(* Logix 5000 project; controller Turck_IOLink_All_Full_AOIs_V0_1 vendor 1 type 14 code 176 rev 32.11; software revision 32.00 *)

TASK MainTask (continuous, watchdog 500 ms) : MainProgram
TASK SafetyTask (periodic, rate 20 ms, priority 10, watchdog 20 ms, safety) : SafetyProgram

MODULES
   Local : vendor 1 type 14 code 176 (Compact 0, rev 32.11)
END_MODULES

TYPE Generic_16_Words :
STRUCT
   Data : INT[16];
END_STRUCT
END_TYPE

TYPE Turck_IOLink_Common_Data :
STRUCT
   Read : BOOL;   // For internal use to integrate IOLRead and IOWrite with IOLService
   Write : BOOL;   // For internal use to integrate IOLRead and IOWrite with IOLService
   Reset : BOOL;   // For internal use to integrate IOLRead and IOWrite with IOLService
   Done : BOOL;   // For internal use to integrate IOLRead and IOWrite with IOLService
   Error : BOOL;   // For internal use to integrate IOLRead and IOWrite with IOLService
   Port_in_Use : SINT;   // Each bit is set to show that a port is in use. If it's not in use the port diagnostics will be disabled so IO-Link can still be used but won't throw a red light if no device plugged
   Port : INT;   // For internal use to integrate IOLRead and IOWrite with IOLService
   Index : INT;   // For internal use to integrate IOLRead and IOWrite with IOLService
   SubIndex : INT;   // For internal use to integrate IOLRead and IOWrite with IOLService
   Length : INT;   // For internal use to integrate IOLRead and IOWrite with IOLService
   TicketNum : INT;   // For internal use to integrate IOLRead and IOWrite with IOLService
   Status : INT;   // For internal use to integrate IOLRead and IOWrite with IOLService
   NextTicketNum : INT;   // For internal use to integrate IOLRead and IOWrite with IOLService
   ReceiveData : SINT[255];   // For internal use to integrate IOLRead and IOWrite with IOLService
   SendData : SINT[145];   // For internal use to integrate IOLRead and IOWrite with IOLService
   Vendor_IDs : INT[8];
   Device_IDs : DINT[8];
   WriteData : DINT;
   Process_Input_Data : Generic_16_Words[8];
   Process_Output_Data : Generic_16_Words[8];
END_STRUCT
END_TYPE

TYPE Universal_IOLink_Info :
STRUCT
   Vendor_Name : STRING;   // Index 16
   Vendor_Text : STRING;   // Index 17
   Product_Name : STRING;   // Index 18
   Product_ID : STRING;   // Index 19
   Product_Text : STRING;   // Index 20
   Serial_Number : STRING;   // Index 21
   Hardware_Revision : STRING;   // Index 22
   Firmware_Revision : STRING;   // Index 23
   Application_Specific_Tag : STRING;   // Index 24
   Function_Tag : STRING;   // Index 25
   Location_Tag : STRING;   // Index 26
   Application_Specific_Tag_Requested : STRING;
END_STRUCT
END_TYPE

ADD_ON_INSTRUCTION Banner_K50_Pro_Advanced_Mode_Full   (* revision 1.0 *)
VAR_INPUT
   Touch_Sensitivity : SINT := 1; {access None}   // Index 82 - Subindex 1 - 0 = Low, 1 = Standard, 2 = High (Default = 1)
   Touch_Function : BOOL;   // Index 82 - Subindex 2 - 0 = Momentary, 1 = Latched
   Touch_Mute_Enable : BOOL;   // Index 82 - Subindex 3 - 0 = Off, 1 = On
   Touch_On_Delay : SINT;   // Index 82 - Subindex 4 - 0-65535 ms
   Custom_Color_1_Red : INT;   // Index 88 - Subindex 1 - 0-255 Amount of Red
   Custom_Color_1_Green : INT;   // Index 88 - Subindex 2 - 0-255 Amount of Green
   Custom_Color_1_Blue : INT;   // Index 88 - Subindex 3 - 0-255 Amount of Blue
   Custom_Color_2_Red : INT;   // Index 89 - Subindex 1 - 0-255 Amount of Red
   Custom_Color_2_Green : INT;   // Index 89 - Subindex 2 - 0-255 - Amount of Green
   Custom_Color_2_Blue : INT;   // Index 89 - Subindex 3 - 0-255 - Amount of Blue
   Port : INT; {required}
END_VAR
VAR_IN_OUT
   Common_Data : Turck_IOLink_Common_Data; {required}
END_VAR
VAR_INPUT
   Animation_Type : SINT; {visible}   // 0 = Off 1 = Steady 2 = Flash 3 = Two Color Flash 4 = 50/50 5 = 50/50 Rotate 6 = Chase 7 = Intensity Sweep 8 = Color Sweep 9 = Sequence
   Animation_Direction : BOOL; {visible}   // 0 = CCW, 1 = CW
   Animation_Pattern : SINT; {visible}   // 0 = Flash, 1 = Strobe, 2 = Three Pulse, 3 = SOS, 4 = Random
   Animation_Speed : SINT; {visible}   // 0 = Slow, 1 = Medium, 2 = Fast, 3 = Custom
   Vibration_Feedback : SINT; {visible}   // 0 = Off, 1 = On, 2 = Animation Pattern
   Dynamic_Sequence : INT; {visible}   // 0-255
   Sequence_Start_Location : SINT; {visible}   // 0 = LED1 1 = LED2 2 = LED3 3 = LED4 4 = LED5 5 = LED6 6 = LED7 7 = LED8
   Color_1 : SINT; {visible}   // 0 = Green 1 = Red 2 = Orange 3 = Amber 4 = Yellow 5 = Lime Green 6 = Spring Green 7 = Cyan 8 = Sky Blue 9 = Blue 10 = Violet 11 = Magenta 12 = Rose 13 = White 14 = Custom1 15 = Custom2
   Color_1_Intensity : SINT; {visible}   // 0 = High, 1 = Medium, 2 = Low, 3 = Off, 4 = Custom
   Color_2 : SINT; {visible}   // 0 = Green 1 = Red 2 = Orange 3 = Amber 4 = Yellow 5 = Lime Green 6 = Spring Green 7 = Cyan 8 = Sky Blue 9 = Blue 10 = Violet 11 = Magenta 12 = Rose 13 = White 14 = Custom1 15 = Custom2
   Color_2_Intensity : SINT; {visible}   // 0 = High, 1 = Medium, 2 = Low, 3 = Off, 4 = Custom
END_VAR
VAR_OUTPUT
   Output_State : BOOL; {access Read Only, visible}   // 0 = Inactive, 1 = Active
   Wrong_or_Missing_Device : BOOL; {access Read Only, visible}
END_VAR
VAR
   Port_Less_One : INT; {access None}
   Port_Bit : SINT; {access None}
   Output_Mode : SINT; {access None}
   Done : DINT; {access None}
   Error : DINT; {access None}
   Active : DINT; {access None}
   Pending : DINT; {access None}
   Pending_or_Active : DINT; {access None}
   Write : DINT; {access None}
   WriteRequest : DINT; {access None}
   Custom_Color_1_Red_Prev : SINT; {access None}
   Custom_Color_1_Green_Prev : SINT; {access None}
   Custom_Color_1_Blue_Prev : SINT; {access None}
   Custom_Color_2_Green_Prev : SINT; {access None}
   StartupDone : BOOL; {access None}
   Read_ONS : DINT; {access None}
   Error_DINT : DINT; {access None}
   StartupCount : DINT; {access None}
   MyTicketNum : DINT[32]; {access None}
   ReadRequest : DINT; {access None}
   DoneCount : DINT; {access None}
   Status : DINT; {access None}
   ErrorCount : DINT; {access None}
   Write_ONS : DINT; {access None}
   Custom_Color_2_Blue_Prev : SINT; {access None}
   Custom_Color_2_Red_Prev : SINT; {access None}
   Device_Connected_ONS : DINT; {access None}
END_VAR

ROUTINE Logic   (* ladder *)
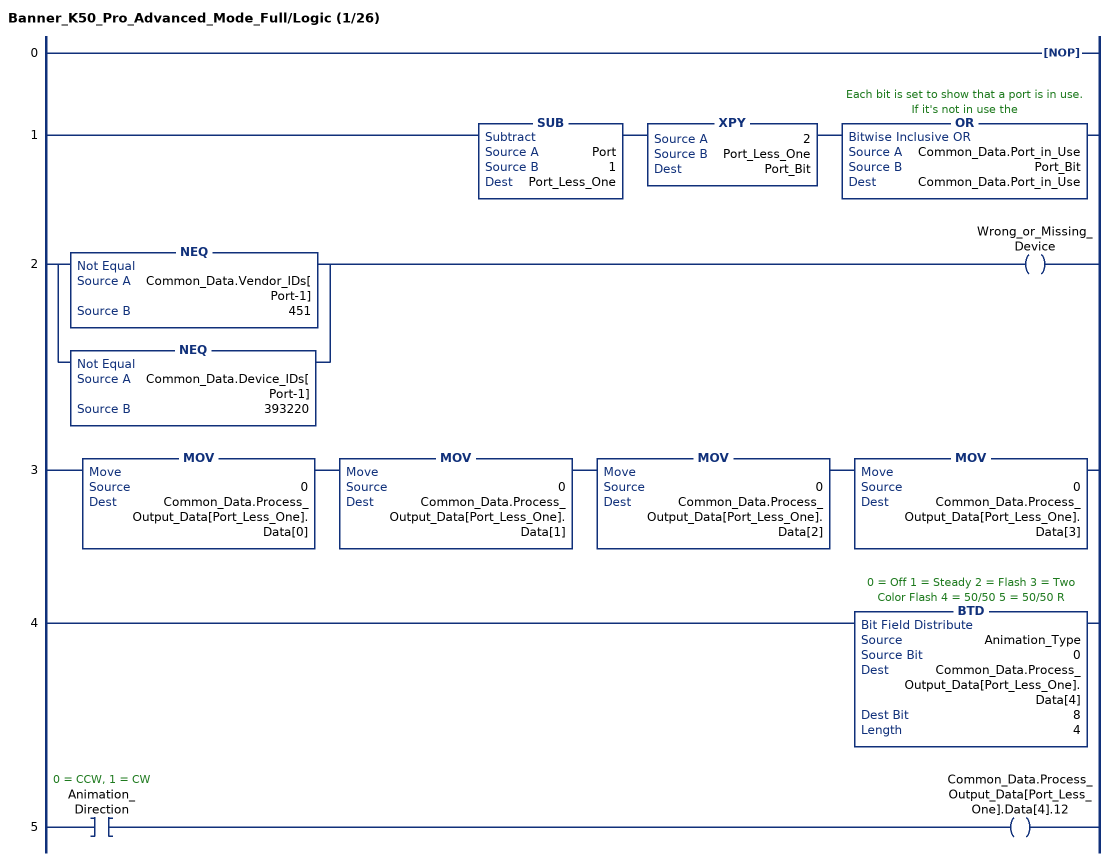
   0: NOP();
   1: SUB(Port,1,Port_Less_One)XPY(2,Port_Less_One,Port_Bit)OR(Common_Data.Port_in_Use,Port_Bit,Common_Data.Port_in_Use);
   2: [NEQ(Common_Data.Vendor_IDs[Port-1],451) ,NEQ(Common_Data.Device_IDs[Port-1],393220) ]OTE(Wrong_or_Missing_Device);
   3: MOV(0,Common_Data.Process_Output_Data[Port_Less_One].Data[0])MOV(0,Common_Data.Process_Output_Data[Port_Less_One].Data[1])MOV(0,Common_Data.Process_Output_Data[Port_Less_One].Data[2])MOV(0,Common_Data.Process_Output_Data[Port_Less_One].Data[3]);
   4: BTD(Animation_Type,0,Common_Data.Process_Output_Data[Port_Less_One].Data[4],8,4);
   5: XIC(Animation_Direction)OTE(Common_Data.Process_Output_Data[Port_Less_One].Data[4].12);
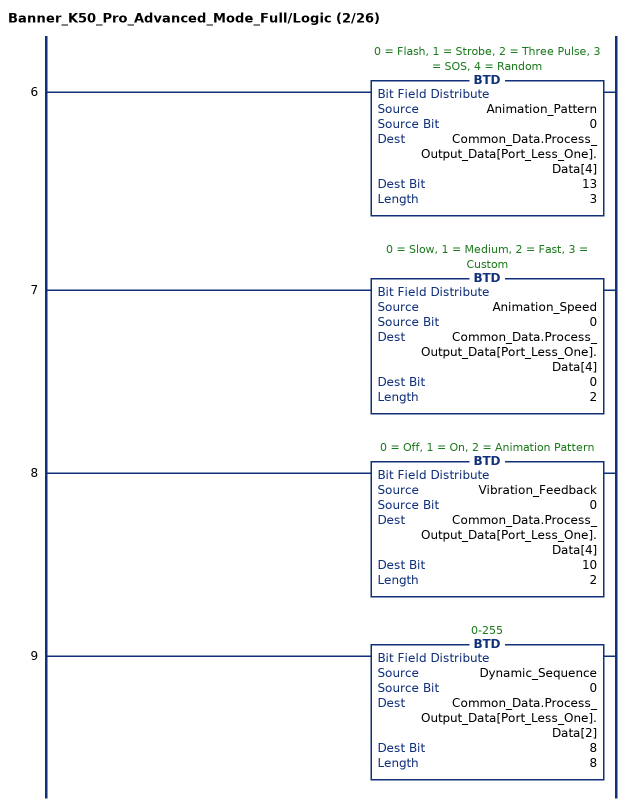
   6: BTD(Animation_Pattern,0,Common_Data.Process_Output_Data[Port_Less_One].Data[4],13,3);
   7: BTD(Animation_Speed,0,Common_Data.Process_Output_Data[Port_Less_One].Data[4],0,2);
   8: BTD(Vibration_Feedback,0,Common_Data.Process_Output_Data[Port_Less_One].Data[4],10,2);
   9: BTD(Dynamic_Sequence,0,Common_Data.Process_Output_Data[Port_Less_One].Data[2],8,8);
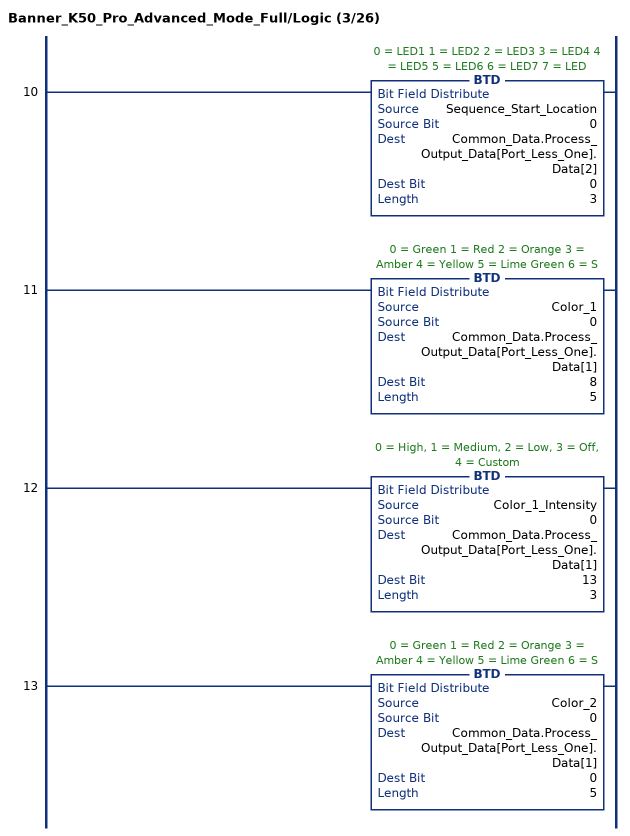
   10: BTD(Sequence_Start_Location,0,Common_Data.Process_Output_Data[Port_Less_One].Data[2],0,3);
   11: BTD(Color_1,0,Common_Data.Process_Output_Data[Port_Less_One].Data[1],8,5);
   12: BTD(Color_1_Intensity,0,Common_Data.Process_Output_Data[Port_Less_One].Data[1],13,3);
   13: BTD(Color_2,0,Common_Data.Process_Output_Data[Port_Less_One].Data[1],0,5);
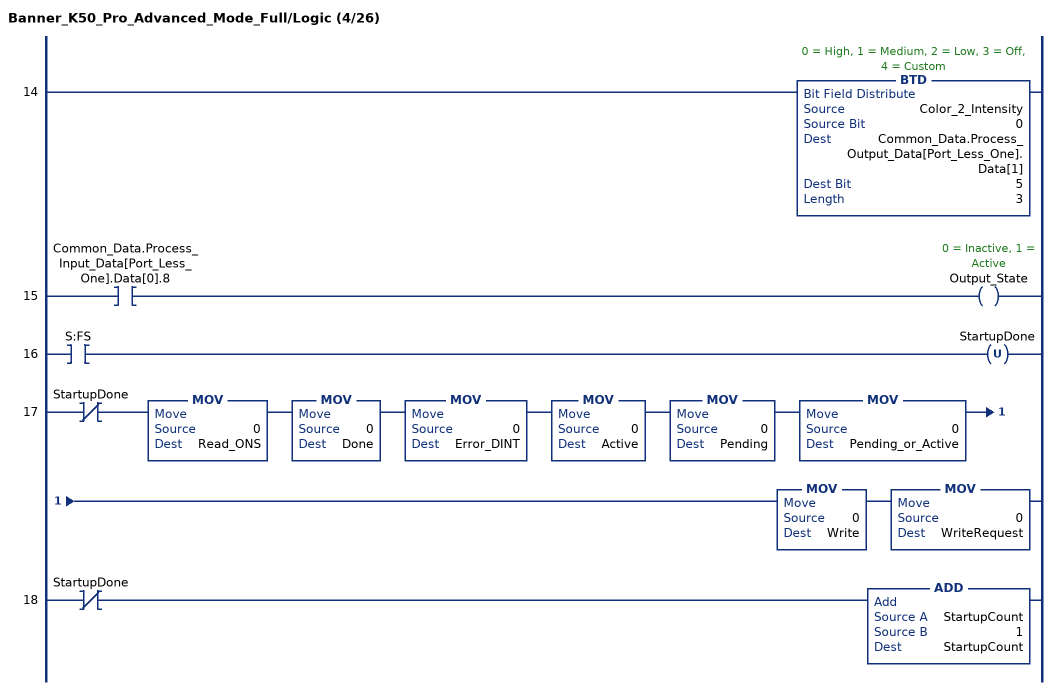
   14: BTD(Color_2_Intensity,0,Common_Data.Process_Output_Data[Port_Less_One].Data[1],5,3);
   15: XIC(Common_Data.Process_Input_Data[Port_Less_One].Data[0].8)OTE(Output_State);
   16: XIC(S:FS)OTU(StartupDone);
   17: XIO(StartupDone)MOV(0,Read_ONS)MOV(0,Done)MOV(0,Error_DINT)MOV(0,Active)MOV(0,Pending)MOV(0,Pending_or_Active)MOV(0,Write)MOV(0,WriteRequest);
   18: XIO(StartupDone)ADD(StartupCount,1,StartupCount);
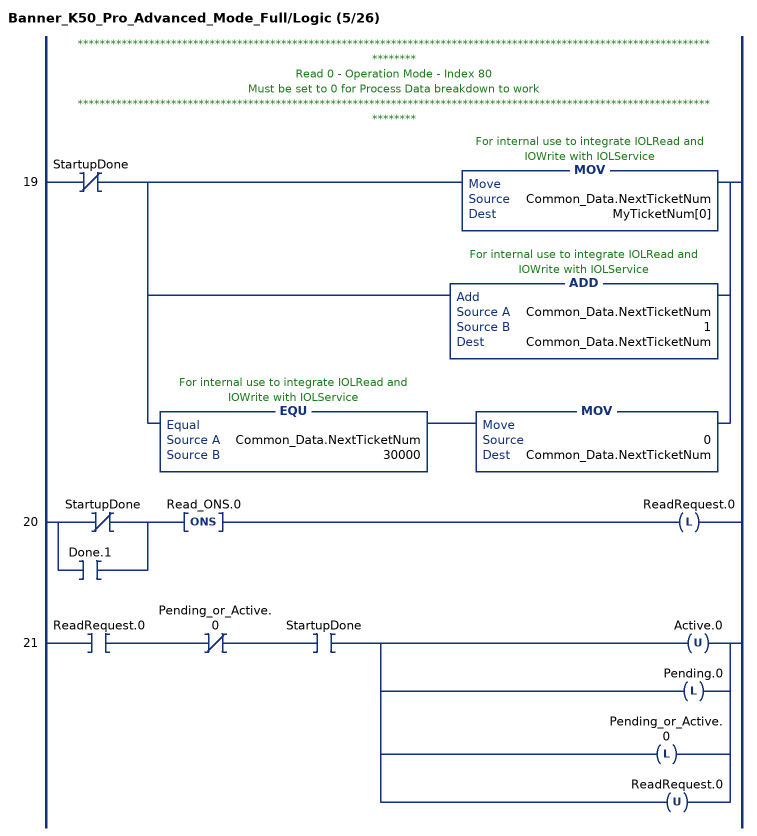
   // ***************************************************************************************************************************
   // Read 0 - Operation Mode - Index 80
   // Must be set to 0 for Process Data breakdown to work
   // ***************************************************************************************************************************
   19: XIO(StartupDone)[MOV(Common_Data.NextTicketNum,MyTicketNum[0]) ,ADD(Common_Data.NextTicketNum,1,Common_Data.NextTicketNum) ,EQU(Common_Data.NextTicketNum,30000) MOV(0,Common_Data.NextTicketNum) ];
   20: [XIO(StartupDone) ,XIC(Done.1) ]ONS(Read_ONS.0)OTL(ReadRequest.0);
   21: XIC(ReadRequest.0)XIO(Pending_or_Active.0)XIC(StartupDone)[OTU(Active.0) ,OTL(Pending.0) ,OTL(Pending_or_Active.0) ,OTU(ReadRequest.0) ];
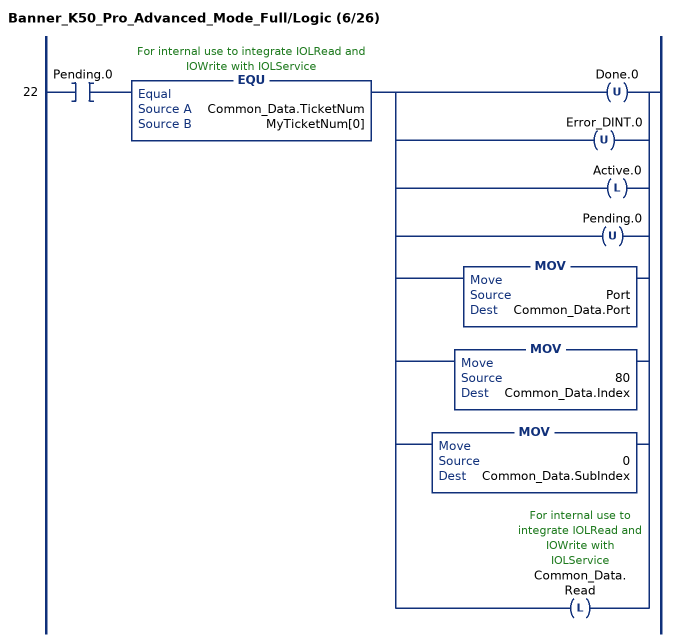
   22: XIC(Pending.0)EQU(Common_Data.TicketNum,MyTicketNum[0])[OTU(Done.0) ,OTU(Error_DINT.0) ,OTL(Active.0) ,OTU(Pending.0) ,MOV(Port,Common_Data.Port) ,MOV(80,Common_Data.Index) ,MOV(0,Common_Data.SubIndex) ,OTL(Common_Data.Read) ];
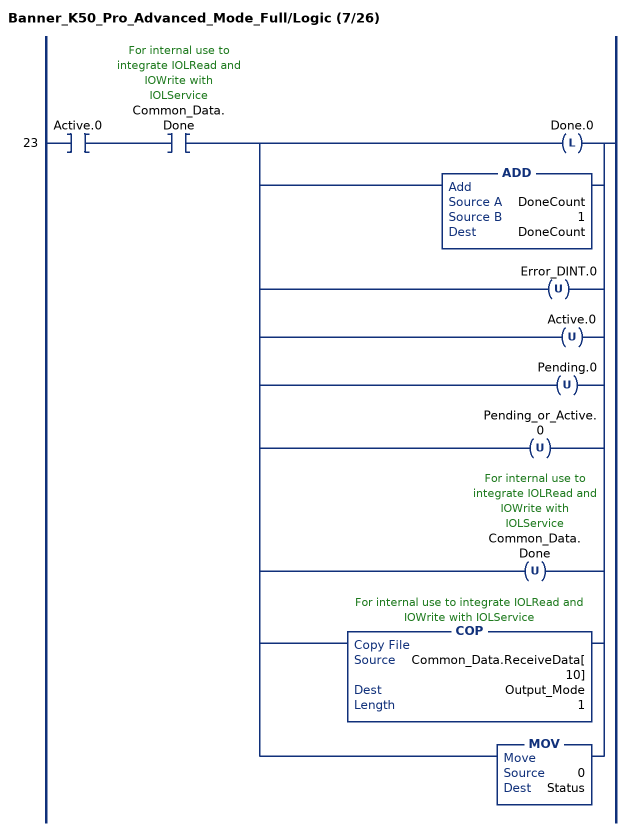
   23: XIC(Active.0)XIC(Common_Data.Done)[OTL(Done.0) ,ADD(DoneCount,1,DoneCount) ,OTU(Error_DINT.0) ,OTU(Active.0) ,OTU(Pending.0) ,OTU(Pending_or_Active.0) ,OTU(Common_Data.Done) ,COP(Common_Data.ReceiveData[10],Output_Mode,1) ,MOV(0,Status) ];
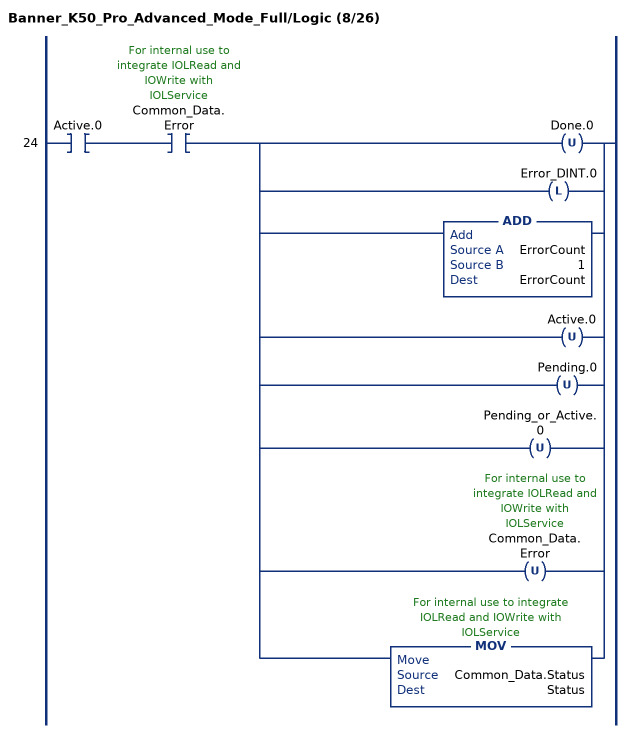
   24: XIC(Active.0)XIC(Common_Data.Error)[OTU(Done.0) ,OTL(Error_DINT.0) ,ADD(ErrorCount,1,ErrorCount) ,OTU(Active.0) ,OTU(Pending.0) ,OTU(Pending_or_Active.0) ,OTU(Common_Data.Error) ,MOV(Common_Data.Status,Status) ];
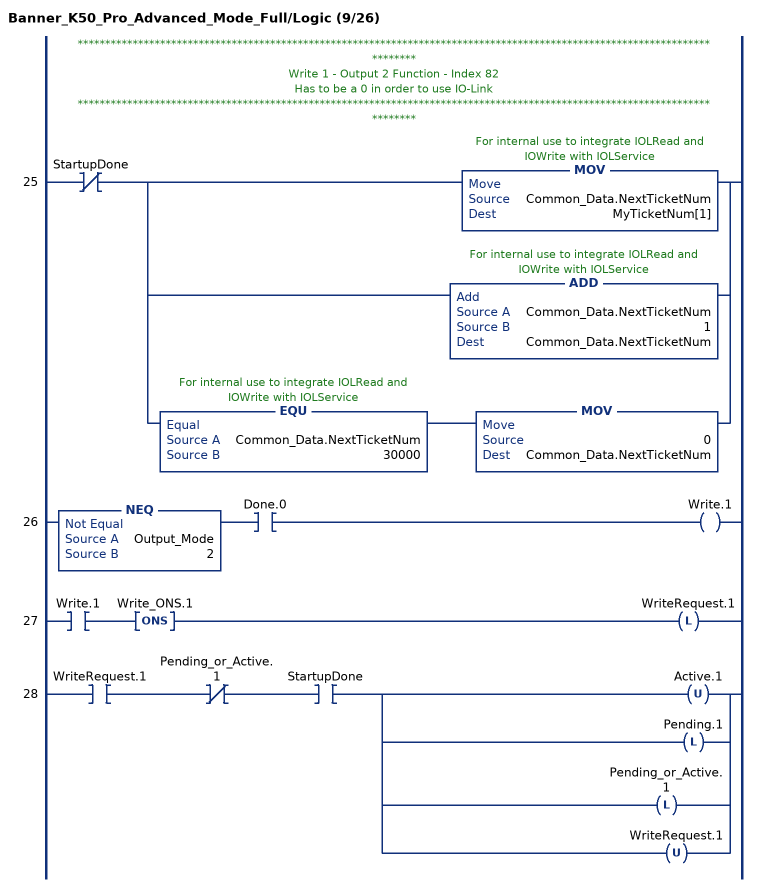
   // ***************************************************************************************************************************
   // Write 1 - Output 2 Function - Index 82
   // Has to be a 0 in order to use IO-Link
   // ***************************************************************************************************************************
   25: XIO(StartupDone)[MOV(Common_Data.NextTicketNum,MyTicketNum[1]) ,ADD(Common_Data.NextTicketNum,1,Common_Data.NextTicketNum) ,EQU(Common_Data.NextTicketNum,30000) MOV(0,Common_Data.NextTicketNum) ];
   26: NEQ(Output_Mode,2)XIC(Done.0)OTE(Write.1);
   27: XIC(Write.1)ONS(Write_ONS.1)OTL(WriteRequest.1);
   28: XIC(WriteRequest.1)XIO(Pending_or_Active.1)XIC(StartupDone)[OTU(Active.1) ,OTL(Pending.1) ,OTL(Pending_or_Active.1) ,OTU(WriteRequest.1) ];
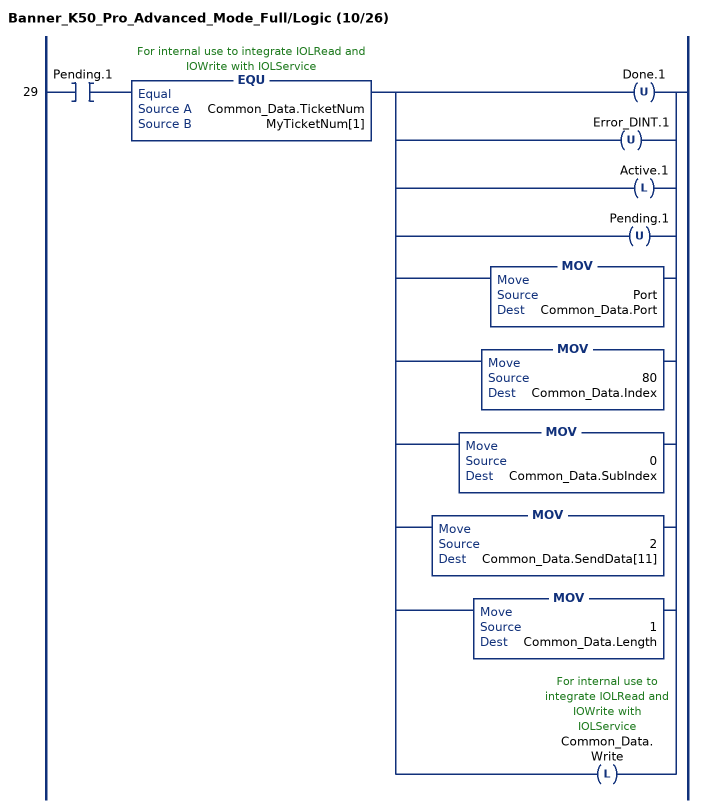
   29: XIC(Pending.1)EQU(Common_Data.TicketNum,MyTicketNum[1])[OTU(Done.1) ,OTU(Error_DINT.1) ,OTL(Active.1) ,OTU(Pending.1) ,MOV(Port,Common_Data.Port) ,MOV(80,Common_Data.Index) ,MOV(0,Common_Data.SubIndex) ,MOV(2,Common_Data.SendData[11]) ,MOV(1,Common_Data.Length) ,OTL(Common_Data.Write) ];
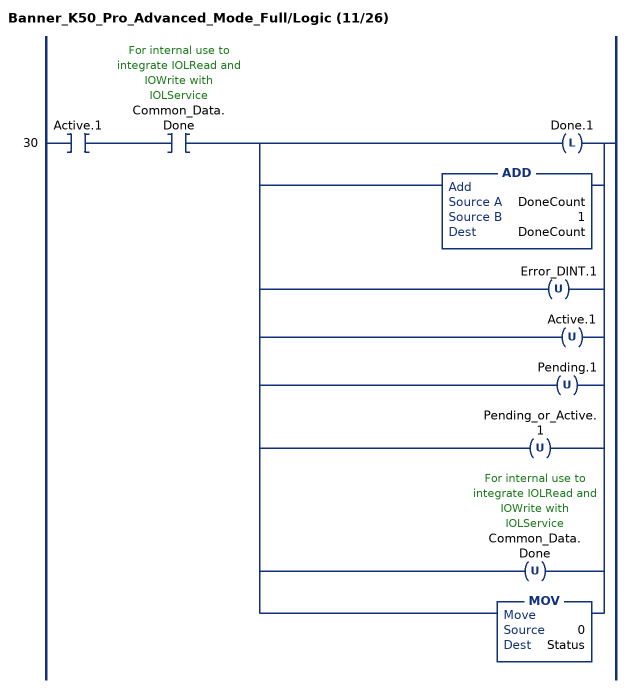
   30: XIC(Active.1)XIC(Common_Data.Done)[OTL(Done.1) ,ADD(DoneCount,1,DoneCount) ,OTU(Error_DINT.1) ,OTU(Active.1) ,OTU(Pending.1) ,OTU(Pending_or_Active.1) ,OTU(Common_Data.Done) ,MOV(0,Status) ];
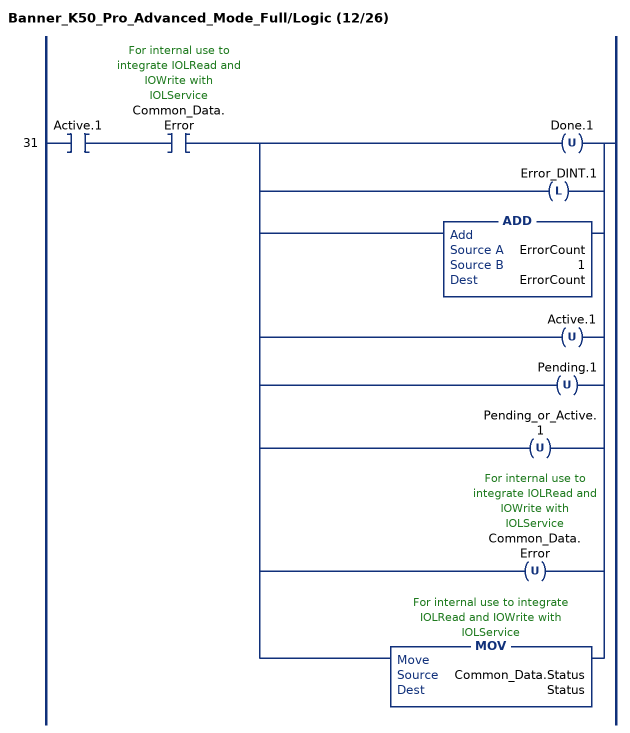
   31: XIC(Active.1)XIC(Common_Data.Error)[OTU(Done.1) ,OTL(Error_DINT.1) ,ADD(ErrorCount,1,ErrorCount) ,OTU(Active.1) ,OTU(Pending.1) ,OTU(Pending_or_Active.1) ,OTU(Common_Data.Error) ,MOV(Common_Data.Status,Status) ];
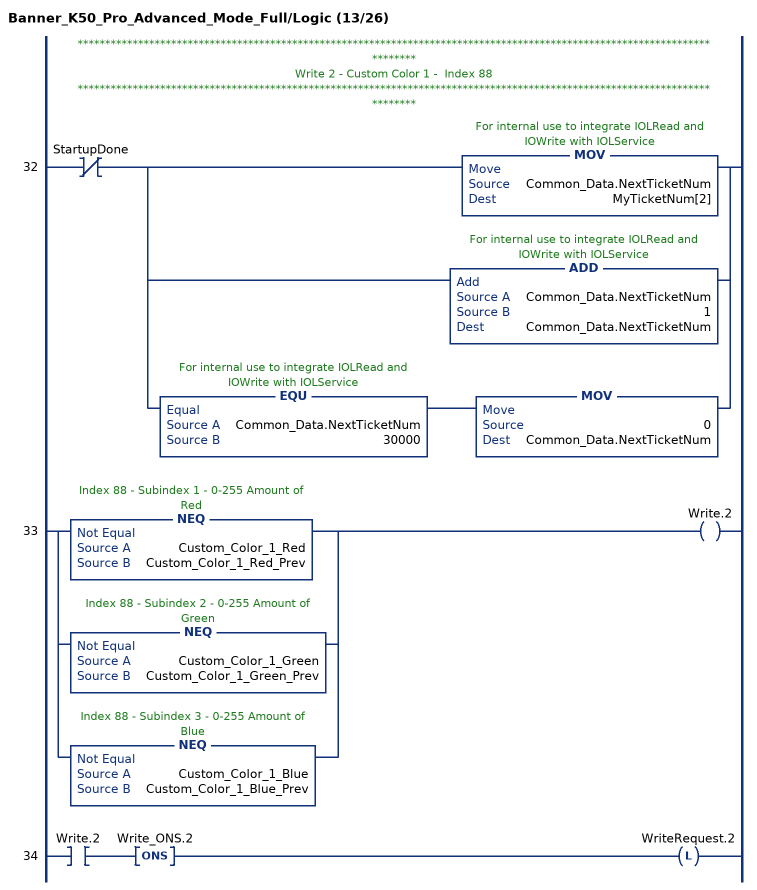
   // ***************************************************************************************************************************
   // Write 2 - Custom Color 1 -  Index 88
   // ***************************************************************************************************************************
   32: XIO(StartupDone)[MOV(Common_Data.NextTicketNum,MyTicketNum[2]) ,ADD(Common_Data.NextTicketNum,1,Common_Data.NextTicketNum) ,EQU(Common_Data.NextTicketNum,30000) MOV(0,Common_Data.NextTicketNum) ];
   33: [NEQ(Custom_Color_1_Red,Custom_Color_1_Red_Prev) ,NEQ(Custom_Color_1_Green,Custom_Color_1_Green_Prev) ,NEQ(Custom_Color_1_Blue,Custom_Color_1_Blue_Prev) ]OTE(Write.2);
   34: XIC(Write.2)ONS(Write_ONS.2)OTL(WriteRequest.2);
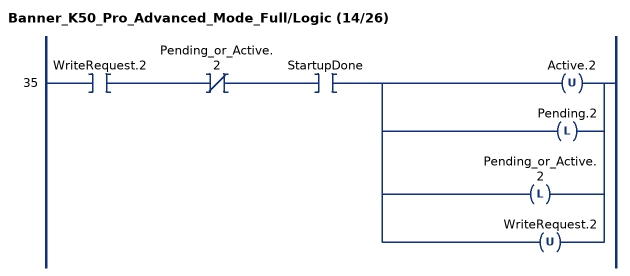
   35: XIC(WriteRequest.2)XIO(Pending_or_Active.2)XIC(StartupDone)[OTU(Active.2) ,OTL(Pending.2) ,OTL(Pending_or_Active.2) ,OTU(WriteRequest.2) ];
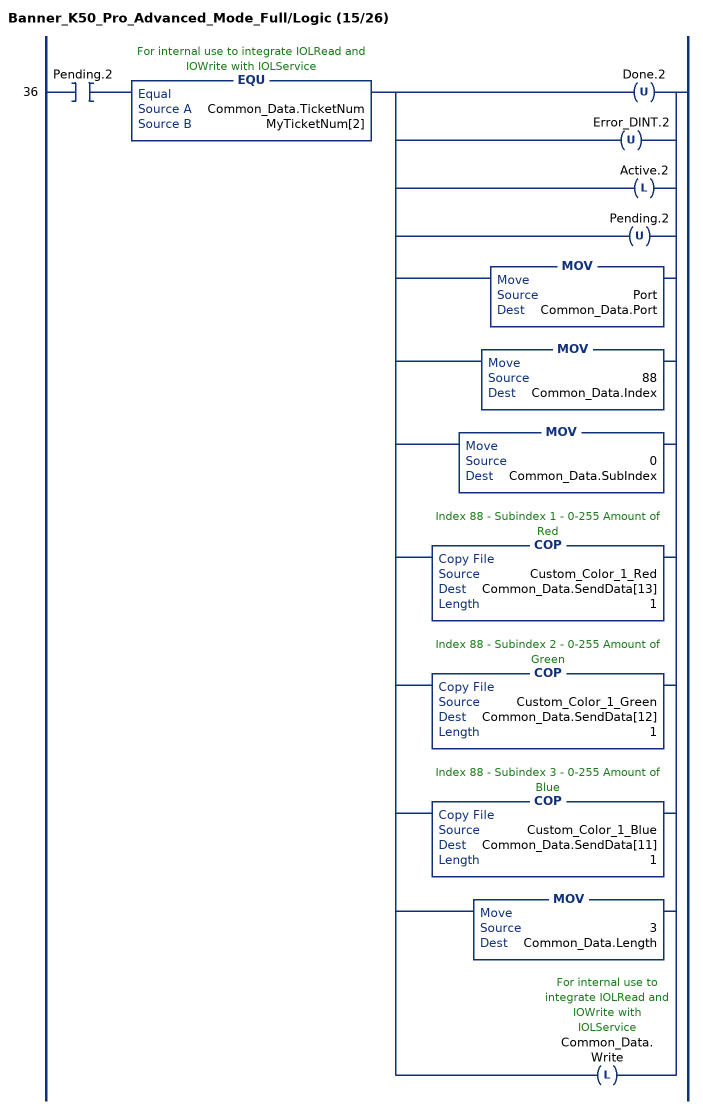
   36: XIC(Pending.2)EQU(Common_Data.TicketNum,MyTicketNum[2])[OTU(Done.2) ,OTU(Error_DINT.2) ,OTL(Active.2) ,OTU(Pending.2) ,MOV(Port,Common_Data.Port) ,MOV(88,Common_Data.Index) ,MOV(0,Common_Data.SubIndex) ,COP(Custom_Color_1_Red,Common_Data.SendData[13],1) ,COP(Custom_Color_1_Green,Common_Data.SendData[12],1) ,COP(Custom_Color_1_Blue,Common_Data.SendData[11],1) ,MOV(3,Common_Data.Length) ,OTL(Common_Data.Write) ];
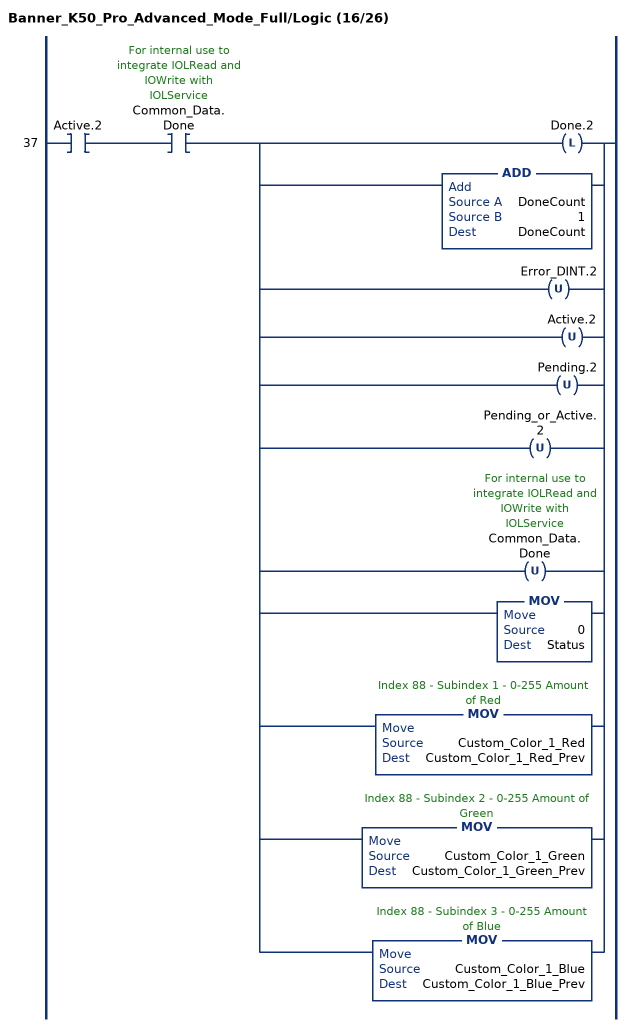
   37: XIC(Active.2)XIC(Common_Data.Done)[OTL(Done.2) ,ADD(DoneCount,1,DoneCount) ,OTU(Error_DINT.2) ,OTU(Active.2) ,OTU(Pending.2) ,OTU(Pending_or_Active.2) ,OTU(Common_Data.Done) ,MOV(0,Status) ,MOV(Custom_Color_1_Red,Custom_Color_1_Red_Prev) ,MOV(Custom_Color_1_Green,Custom_Color_1_Green_Prev) ,MOV(Custom_Color_1_Blue,Custom_Color_1_Blue_Prev) ];
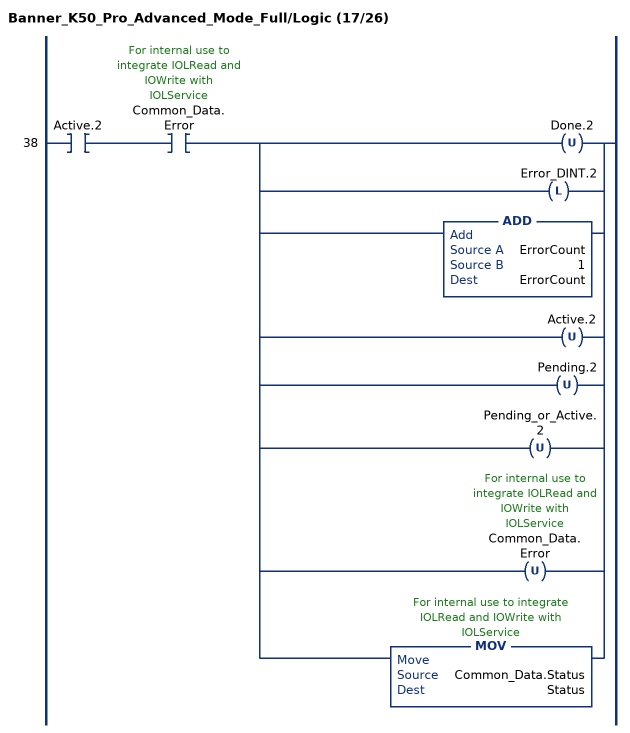
   38: XIC(Active.2)XIC(Common_Data.Error)[OTU(Done.2) ,OTL(Error_DINT.2) ,ADD(ErrorCount,1,ErrorCount) ,OTU(Active.2) ,OTU(Pending.2) ,OTU(Pending_or_Active.2) ,OTU(Common_Data.Error) ,MOV(Common_Data.Status,Status) ];
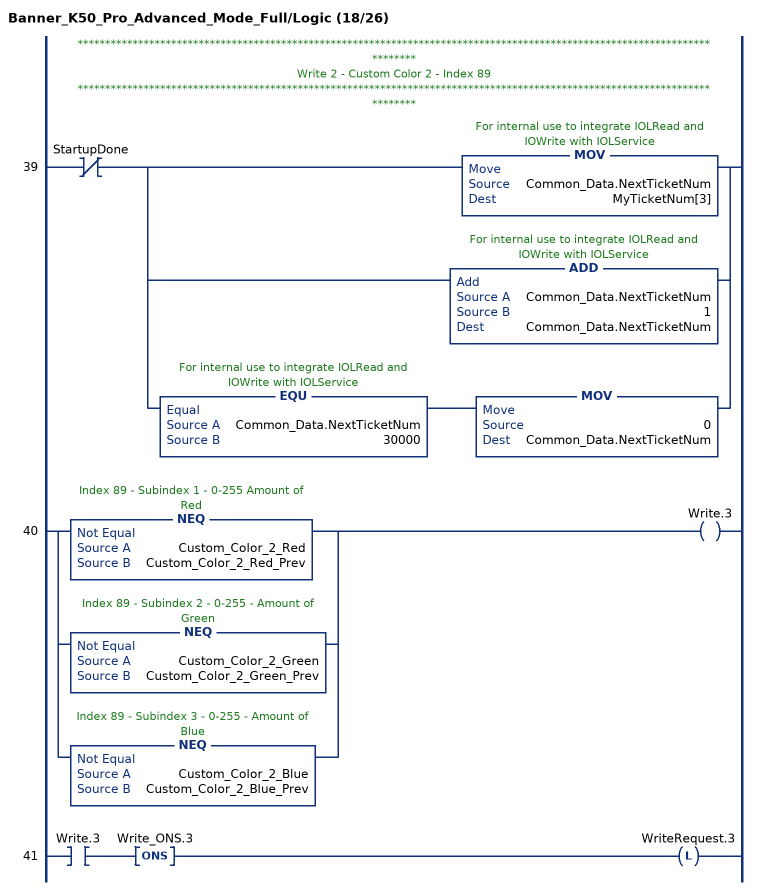
   // ***************************************************************************************************************************
   // Write 2 - Custom Color 2 - Index 89
   // ***************************************************************************************************************************
   39: XIO(StartupDone)[MOV(Common_Data.NextTicketNum,MyTicketNum[3]) ,ADD(Common_Data.NextTicketNum,1,Common_Data.NextTicketNum) ,EQU(Common_Data.NextTicketNum,30000) MOV(0,Common_Data.NextTicketNum) ];
   40: [NEQ(Custom_Color_2_Red,Custom_Color_2_Red_Prev) ,NEQ(Custom_Color_2_Green,Custom_Color_2_Green_Prev) ,NEQ(Custom_Color_2_Blue,Custom_Color_2_Blue_Prev) ]OTE(Write.3);
   41: XIC(Write.3)ONS(Write_ONS.3)OTL(WriteRequest.3);
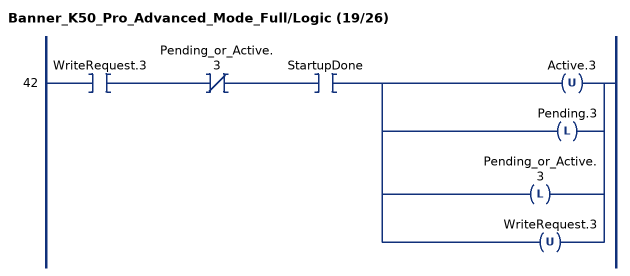
   42: XIC(WriteRequest.3)XIO(Pending_or_Active.3)XIC(StartupDone)[OTU(Active.3) ,OTL(Pending.3) ,OTL(Pending_or_Active.3) ,OTU(WriteRequest.3) ];
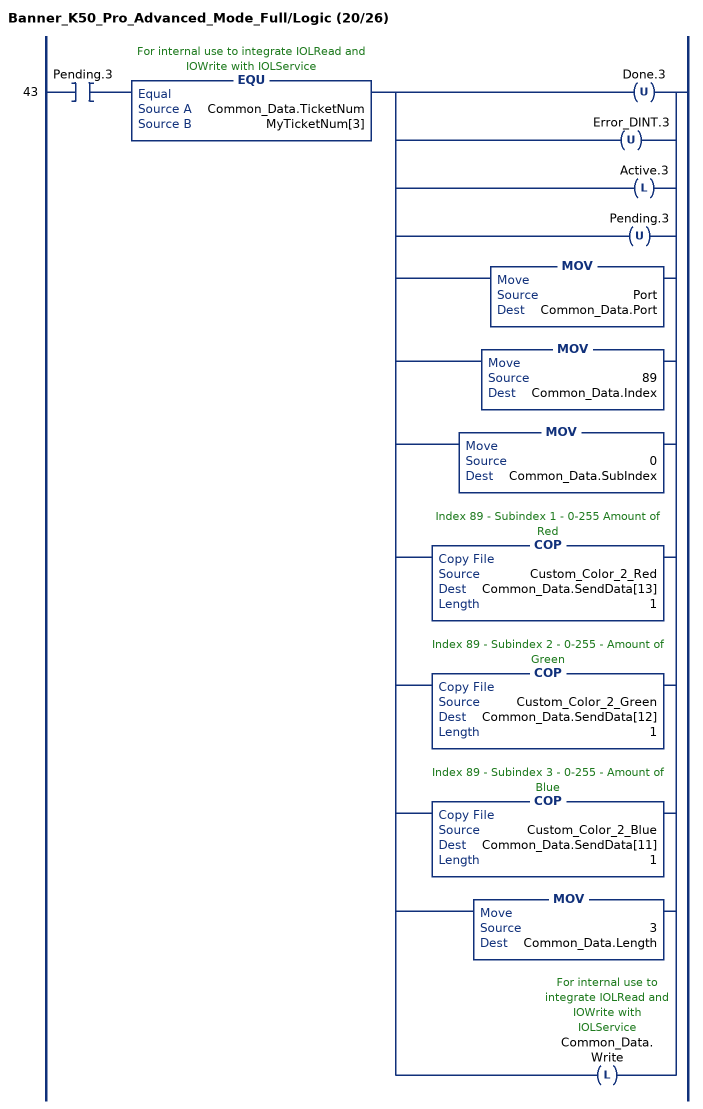
   43: XIC(Pending.3)EQU(Common_Data.TicketNum,MyTicketNum[3])[OTU(Done.3) ,OTU(Error_DINT.3) ,OTL(Active.3) ,OTU(Pending.3) ,MOV(Port,Common_Data.Port) ,MOV(89,Common_Data.Index) ,MOV(0,Common_Data.SubIndex) ,COP(Custom_Color_2_Red,Common_Data.SendData[13],1) ,COP(Custom_Color_2_Green,Common_Data.SendData[12],1) ,COP(Custom_Color_2_Blue,Common_Data.SendData[11],1) ,MOV(3,Common_Data.Length) ,OTL(Common_Data.Write) ];
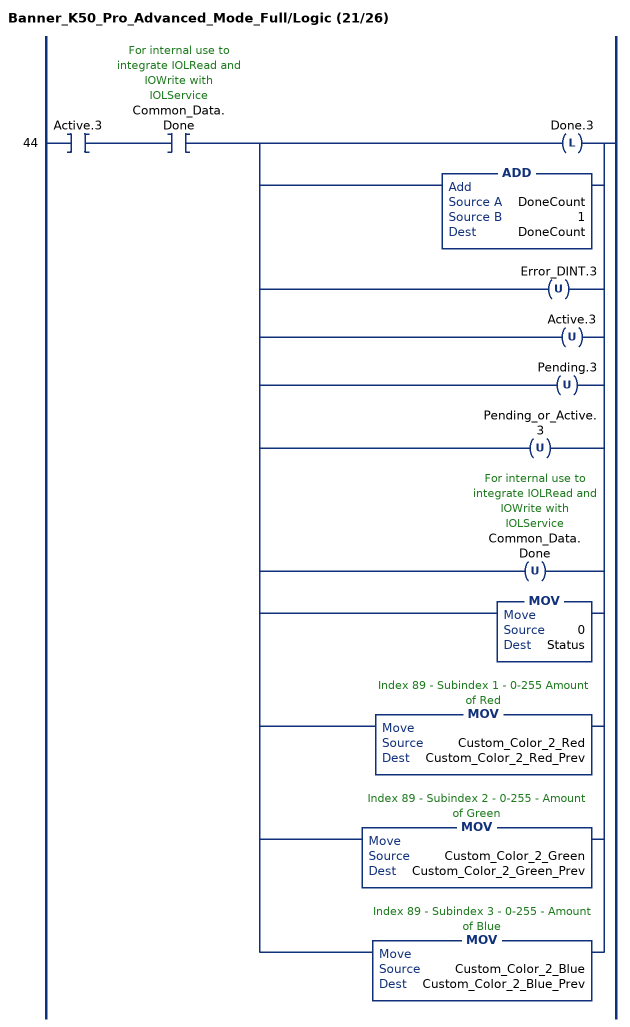
   44: XIC(Active.3)XIC(Common_Data.Done)[OTL(Done.3) ,ADD(DoneCount,1,DoneCount) ,OTU(Error_DINT.3) ,OTU(Active.3) ,OTU(Pending.3) ,OTU(Pending_or_Active.3) ,OTU(Common_Data.Done) ,MOV(0,Status) ,MOV(Custom_Color_2_Red,Custom_Color_2_Red_Prev) ,MOV(Custom_Color_2_Green,Custom_Color_2_Green_Prev) ,MOV(Custom_Color_2_Blue,Custom_Color_2_Blue_Prev) ];
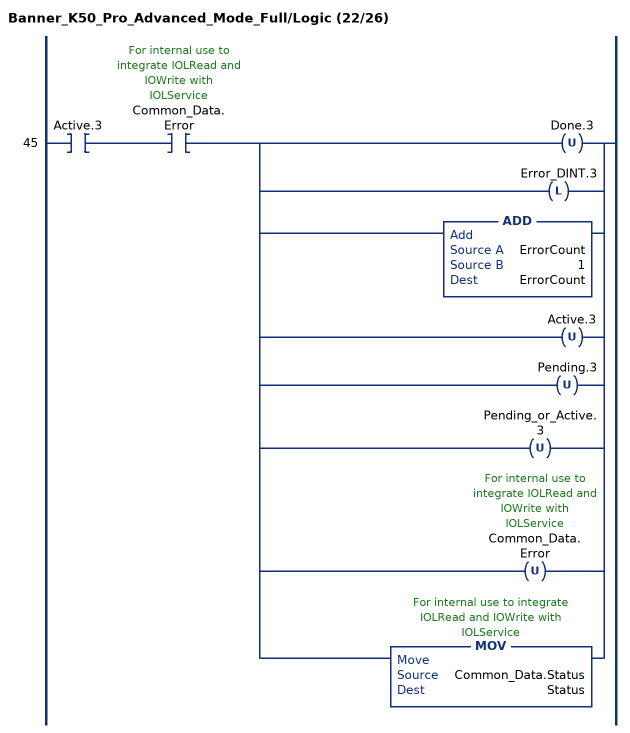
   45: XIC(Active.3)XIC(Common_Data.Error)[OTU(Done.3) ,OTL(Error_DINT.3) ,ADD(ErrorCount,1,ErrorCount) ,OTU(Active.3) ,OTU(Pending.3) ,OTU(Pending_or_Active.3) ,OTU(Common_Data.Error) ,MOV(Common_Data.Status,Status) ];
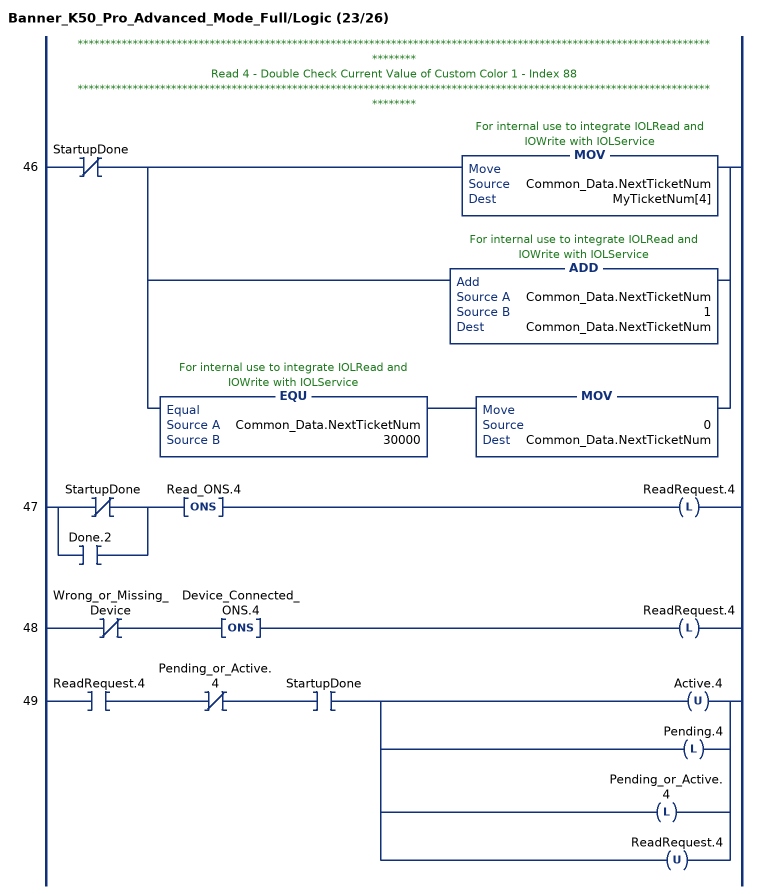
   // ***************************************************************************************************************************
   // Read 4 - Double Check Current Value of Custom Color 1 - Index 88
   // ***************************************************************************************************************************
   46: XIO(StartupDone)[MOV(Common_Data.NextTicketNum,MyTicketNum[4]) ,ADD(Common_Data.NextTicketNum,1,Common_Data.NextTicketNum) ,EQU(Common_Data.NextTicketNum,30000) MOV(0,Common_Data.NextTicketNum) ];
   47: [XIO(StartupDone) ,XIC(Done.2) ]ONS(Read_ONS.4)OTL(ReadRequest.4);
   48: XIO(Wrong_or_Missing_Device)ONS(Device_Connected_ONS.4)OTL(ReadRequest.4);
   49: XIC(ReadRequest.4)XIO(Pending_or_Active.4)XIC(StartupDone)[OTU(Active.4) ,OTL(Pending.4) ,OTL(Pending_or_Active.4) ,OTU(ReadRequest.4) ];
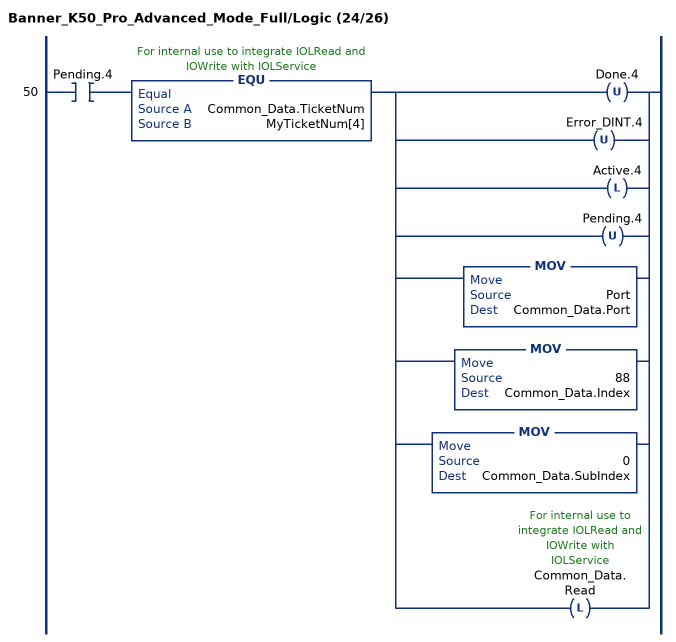
   50: XIC(Pending.4)EQU(Common_Data.TicketNum,MyTicketNum[4])[OTU(Done.4) ,OTU(Error_DINT.4) ,OTL(Active.4) ,OTU(Pending.4) ,MOV(Port,Common_Data.Port) ,MOV(88,Common_Data.Index) ,MOV(0,Common_Data.SubIndex) ,OTL(Common_Data.Read) ];
